    // Command processing
    IF #fbInputs.Cmd_Stop THEN
        // STOP: controlled stop without generating an error + return to safe position
        #bPauseActive := FALSE;
        #bStartSeq := FALSE;
        // Drop every other axis-motion trigger before handing the axes to the STOPPING
        // park move. Without this, a Stop pressed during a clearance/park move (13/16) or
        // during the homing sequence (15) leaves fbMoveX/Z_HomeClr or fbHomeX/Z/Tool
        // executing while fbMoveX/Z_Stop is also commanded -- two MC_ function blocks
        // fighting for the same axis. Latent before the sheet-load park change; state 16
        // is now on the normal cycle path (every reposition), so it is reachable in
        // routine operation rather than only mid-homing.
        #bHomeClrX := FALSE; #bHomeClrZ := FALSE;
        #bHomeXExec := FALSE; #bHomeZExec := FALSE; #bHomeToolExec := FALSE;
        #homeSeqState := 0;
        // If running, go to special STOP sequence; otherwise go directly to STOPPED
        IF (#State >= STATE_STARTING AND #State < STATE_ERROR AND #State <> 100) OR (#State = STATE_PAUSED) THEN
            #State := STATE_STOPPING;
        ELSE
            #State := STATE_STOPPED;
        END_IF;
    END_IF;
    // Reset and Restart are blocked while E-Stop is active.
    // Operator must physically release E-Stop before clearing any error state.
    IF #fbInputs.Cmd_Reset AND (#EStop_OK OR "DB_HMI".Bypass_EStop) THEN
        #bDoHardReset := TRUE;
    END_IF;

    // Btn_Restart - restart program from beginning (from ERROR or PAUSED).
    // This block fires BEFORE the CASE state machine, so CASE 999/25 restart handlers
    // are bypassed. All required cleanup must be done here.
    IF #restartEdge AND (#State = STATE_ERROR OR #State = STATE_PAUSED)
       AND (#EStop_OK OR "DB_HMI".Bypass_EStop) THEN
        #State := STATE_STOPPED;
        #bPauseActive := FALSE;
        #Error := FALSE;
        #bResetRecipe := TRUE;      // Reset recipe handler to IDLE (was missing -- bug fix)
        #prevSafetyError := FALSE;  // Fresh safety evaluation on restart
        #savedLineIndex := -1;
        #savedProgram := -1;
        "DB_HMI".ResumeLine := -1;
        IF NOT "DB_MachineConfig".Bypass_MandrelLock THEN
            #bMandrelRetractPending := TRUE;  // ITEM-32: deferred — spindle may still be spinning; wait SpindleStopSafeTime
        END_IF;
        #fbAlarmManager(NewError := FALSE, NewErrorCode := 0,
                        AcknowledgeError := TRUE);  // Clear active alarm (was missing -- bug fix)
    END_IF;

    // Pause - one-shot SET only (no toggle). Only Btn_Continue resumes.
    IF #fbInputs.Cmd_Pause AND #Running AND NOT #bPauseActive THEN #bPauseActive := TRUE; END_IF;

    #Running := (#State >= 10) AND (#State < STATE_ERROR);
    #IsPaused := (#State = STATE_PAUSED);

    // Update HMI status lamps
    "DB_HMI".IsRunning := #Running;
    "DB_HMI".IsPaused := #IsPaused;
    "DB_HMI".HasError := (#State = STATE_ERROR);

    // Warning: only E-Stop bypass is shown on HMI (Door/Air/Drive bypasses silently permitted for setup)
    // Since 2026-08-12 the bypass no longer blocks auto start, so this banner is the
    // ONLY indication that the machine will run with the E-Stop circuit defeated.
    // WarningID stays 1 (WinCC text list key); the wording changed -- keep
    // tools/hmi_texts.csv row 'warning,1' in step with this string.
    // Priority chain, highest first. E-Stop bypass is never suppressed by anything --
    // it is the only sign that the machine will run unguarded, so it outranks a
    // transient interlock message. A blocked tool jog therefore shows no banner while
    // the bypass is on; the jog is still refused, which is the part that matters.
    "DB_HMI".HasWarning := "DB_HMI".Bypass_EStop OR #bToolAxisBlocked
                           OR #bToolStepBlocked OR #bBlindMoveBlocked;
    IF "DB_HMI".Bypass_EStop THEN
        "DB_HMI".WarningText    := 'DANGER: E-Stop bypassed - machine runs unguarded';
        "DB_HMI".WarningID      := 1;
    ELSIF #bToolAxisBlocked OR #bToolStepBlocked THEN
        // Shown as soon as the tool axis is selected with the lock engaged, not only
        // after a button press: the operator learns why before pushing, and the
        // message explains the refusal if they push anyway. No latch, no timer --
        // it clears itself when the lock releases or another axis is selected.
        // The turret-step buttons (#bToolStepBlocked) have no "selection" to hook, so
        // for them the banner is necessarily press-driven and shares WarningID 3 --
        // same cause, same wording, no new text-list row needed.
        "DB_HMI".WarningText    := 'Tool axis locked - ToolHeadLock is engaged';
        "DB_HMI".WarningID      := 3;
    ELSIF #bBlindMoveBlocked THEN
        // ITEM-56d: MoveAbsolute / GoSafe / GoZero are refused while halted in a PNP zone.
        // A dead button with no explanation is how an operator concludes the panel is broken,
        // so say why and name the two things that DO work. Warning, not an error -- a refused
        // button must never demand a Reset (same rule as the ToolHeadLock interlock above).
        // #bBlindMoveBlocked is assigned near the bottom of this FB, so this reads the previous
        // scan's value; harmless, because STATE_PNP_HALT is held for many scans.
        "DB_HMI".WarningText    := 'Blocked in proximity zone - use jog or Home to escape';
        "DB_HMI".WarningID      := 4;
    ELSE
        "DB_HMI".WarningText    := '';
        "DB_HMI".WarningID      := 0;
    END_IF;

    // Update HMI status message based on state (English only since 2026-08-10 --
    // Spanish comes from a WinCC text list keyed off DB_HMI.MachineState, ITEM-55)
    CASE #State OF
        0:   "DB_HMI".StatusMsg := 'Stopped';
        5:   "DB_HMI".StatusMsg := 'Manual Mode';
        10:  "DB_HMI".StatusMsg := 'Starting...';
        11:  "DB_HMI".StatusMsg := 'Loading recipe...';
        12:  "DB_HMI".StatusMsg := 'Pre-scanning...';
        13:  "DB_HMI".StatusMsg := 'Clearing PNP zone...';
        14:  "DB_HMI".StatusMsg := 'Waiting for sheet...';
        15:  "DB_HMI".StatusMsg := 'Homing...';
        16:  "DB_HMI".StatusMsg := 'Sheet-load park move...';
        17:  "DB_HMI".StatusMsg := 'Lock engaging...';
        18:  "DB_HMI".StatusMsg := 'Stopping...';
        29:  "DB_HMI".StatusMsg := 'Lock releasing...';
        19:  "DB_HMI".StatusMsg := 'Homing (post-stop)...';
        20:  "DB_HMI".StatusMsg := 'Running';
        21:  "DB_HMI".StatusMsg := 'Returning to zero...';
        22:  "DB_HMI".StatusMsg := 'PNP Halt - jog to escape limit zone';
        25:  "DB_HMI".StatusMsg := 'Paused';
        30:  "DB_HMI".StatusMsg := 'Tool Change';
        35:  "DB_HMI".StatusMsg := 'Tool Change Wait';
        100: "DB_HMI".StatusMsg := 'Program Complete';
        999: "DB_HMI".StatusMsg := 'ERROR';
    END_CASE;

    // =========================================================================
    // ALARM MANAGER - call FIRST so outputs are ready for DB_HMI
    // =========================================================================
    // NOTE: Acknowledge is done only on edge (ackEdge), not level.
    // This keeps ActiveError/HMI bools visible until the operator actually presses Ack.
    //
    // Error_ProcessState: captured HERE, guarded, and nowhere else (2026-08-17). It used
    // to be assigned #State unconditionally a few lines below, every scan -- which made it
    // a duplicate of DB_Diagnostic.Process_State and destroyed the thing it was named for.
    // Every diagnostic doc read it as "the state the machine was in when it faulted"; it
    // never held that. One guard here covers all ~30 alarm sites, because they all funnel
    // through #newErrorFlag. Do not add a second writer -- the two that existed
    // (STATE_ERROR in this file, FB_RecipeHandler state 999) both wrote a constant.
    IF #newErrorFlag THEN
        "DB_Diagnostic".Error_ProcessState := #State;
    END_IF;

    #fbAlarmManager(NewError         := #newErrorFlag,
                    NewErrorCode     := #newErrorCode,
                    AcknowledgeError := #ackEdge OR #fbInputs.Cmd_Reset,
                    ActiveProgram    := #activeProgram,
                    ActiveLine       := #fbRecipeHandler.CurrentLine);  // ITEM-26
    #newErrorFlag := FALSE;

    // Debug helpers: copy alarm/diagnostic info into DB_Diagnostic for easy tracing
    // This ensures a snapshot of the latest active error code is always visible for debugging.
    // (Error_ProcessState is NOT written here any more -- see the guarded capture above.
    //  The live state is DB_Diagnostic.Process_State, written at the bottom of this FB.)
    "DB_Diagnostic".Error_Code := #fbAlarmManager.ActiveErrorCode;
    // If recipe reported a line error, keep that; otherwise -1
    IF "DB_Diagnostic".Error_Line < 0 THEN
        "DB_Diagnostic".Error_Line := -1;
    END_IF;

    // Copy alarm outputs to HMI (now reads CURRENT scan values)
    "DB_HMI".ErrorID       := #fbAlarmManager.ActiveErrorCode;
    "DB_HMI".ErrorText     := #fbAlarmManager.ActiveErrorText;
    // ITEM-08: If no active alarm text but a safety condition is blocking, show it.
    // This covers the case where the operator is in STOPPED state with door open / E-Stop active
    // after a previous error was acknowledged — AlarmManager cleared its text but the safety
    // condition is still live and writing to DB_Diagnostic.Error_Text.
    // Use compact customer-facing text here; DB_Diagnostic keeps the developer detail.
    // ITEM-16: ErrorDetail is also written here so the operator does not need DB_Diagnostic.
    IF "DB_HMI".ErrorText = '' AND NOT #fbSafetyMonitor.SafeToRun THEN
        CASE #fbSafetyMonitor.ErrorCode OF
            16#0401: "DB_HMI".ErrorText      := 'EMERGENCY STOP active';
                     "DB_HMI".ErrorDetail    := 'Check E-Stop pushbutton and wiring';
            16#0402: "DB_HMI".ErrorText      := 'Safety door open';
                     "DB_HMI".ErrorDetail    := 'Close the safety door to continue';
            16#0403: "DB_HMI".ErrorText      := 'Drives not ready';
                     "DB_HMI".ErrorDetail    := 'Check contactor, enable wiring and drive status';
            16#0404: "DB_HMI".ErrorText      := 'Air pressure low';
                     "DB_HMI".ErrorDetail    := 'Check air compressor and pressure switch';
            ELSE:    "DB_HMI".ErrorText      := 'Safety interlock active';
                     "DB_HMI".ErrorDetail    := '';
        END_CASE;
    END_IF;
    "DB_HMI".CurrentTool := #CurrentTool;

    // Reset TO errors (only on AckError or full reset)
    // BUG FIX: MC_Reset is triggered only by edge signals. Btn_AckError level signal
    // is not used -- when the button is held, Execute stays HIGH continuously, which
    // adversely affects TO error management (new errors may be masked).
    #fbResetX(Execute := #ackEdge OR #fbInputs.Cmd_Reset, Axis := #Axis_X);
    #fbResetZ(Execute := #ackEdge OR #fbInputs.Cmd_Reset, Axis := #Axis_Z);
    #fbResetTool(Execute := #ackEdge OR #fbInputs.Cmd_Reset, Axis := #Axis_Tool);
    #fbResetSpindle(Execute := #ackEdge OR #fbInputs.Cmd_Reset, Axis := #Axis_Spindle);

    // =========================================================================
    // HARD RESET
    // =========================================================================
    // Single place that defines what a full reset clears.
    // Triggered from exactly two places:
    //   1. bInitDone block (first PLC scan after power-up / warm restart)
    //   2. Cmd_Reset handler (operator presses Reset button)
    // Motion-FB execute flags (bHomeXExec, bStopMoveX, etc.) are cleared by the
    // STATE_STOPPED CASE block which runs on this same scan right after this block.
    IF #bDoHardReset THEN
        // Reference validity -- evaluated FIRST, while #State still holds the state the
        // operator pressed Reset in (the assignment below overwrites it).
        //
        // This used to be an unconditional #bRequireHoming := TRUE at the bottom of the block,
        // which made every Reset cost a full homing cycle on the next auto start. Operators
        // press Reset out of habit, often several times, from an idle machine — where nothing
        // has happened that could invalidate the reference. Now only a reset pressed from a
        // state where an axis could have been moving arms the latch, because #bHaltAllAxes
        // above aborts whatever was in progress.
        //
        // WHITELIST, not blacklist: anything not listed counts as "could have been moving", so
        // a state added later fails safe. The three listed states are motionless by definition:
        //   STOPPED (0)  — idle
        //   MANUAL  (5)  — jogging is tracked by the TO, and STATE_STARTING already handles
        //                  "trusted but parked elsewhere" with a park move. An MC_Home aborted
        //                  mid-seek in manual clears StatusBits.HomingDone by itself, and
        //                  bRefTrusted checks that separately
        //   COMPLETE(100)— program finished, axes parked
        // This NEVER clears the latch — only ever sets it — so a homing requirement raised
        // earlier by an E-Stop, a fault or loss of drive power survives any number of resets.
        IF NOT (#State = STATE_STOPPED OR #State = STATE_MANUAL OR #State = 100) THEN
            #bRequireHoming := TRUE;
        END_IF;
        #bHaltAllAxes    := TRUE;   // ITEM-31: abort any in-progress MC_Home before clearing state
        #State           := STATE_STOPPED;
        #Error           := FALSE;
        #bPauseActive    := FALSE;
        #bResumeSpeedup  := FALSE;   // Cancel any pending pause spin-up wait
        #bResumeLockChk  := FALSE;   // Cancel any pending pause lock verification
        #savedLineIndex  := -1;
        #savedProgram    := -1;
        "DB_HMI".ResumeLine := -1;
        #prevSafetyError := FALSE;
        #bResetRecipe                := TRUE;
        #bRecipeLoadExec             := FALSE;  // drop READ_DBL REQ. fbRecipeLoader.Reset is driven
                                                // by bResetRecipe (set TRUE just above) at its call
                                                // site -- NOT by bDoHardReset, which is cleared at
                                                // the end of this block and would never be seen
                                                // there. That Reset also clears LoadedProgram ->
                                                // forces a fresh copy before the next cycle
        #bSheetWaitPhase2            := FALSE;
        #bSheetWaitPhase3            := FALSE;
        IF NOT "DB_MachineConfig".Bypass_MandrelLock THEN
            #bMandrelRetractPending  := TRUE;   // ITEM-32: deferred — machine may have been RUNNING; wait SpindleStopSafeTime
        END_IF;
        #bSheetHolderRetractHold     := TRUE;   // Release sheet holder regardless of which state was active.
                                                // TRUE (not FALSE) is the safe hard-reset default: this latch
                                                // commands the retract, and the blocked centre will otherwise
                                                // hold the piston wherever the fault left it.
                                                // tonSheetHolderHold needs no explicit reset: its IN is this
                                                // latch, so setting it TRUE here restarts the window cleanly.
        // BackSupport end-of-recipe retract (ITEM-41): deliberately NOT reset here, and the edge
        // memory is deliberately NOT seeded here. Same class of exception as
        // #bMandrelRetractPending above -- an in-flight safety motion outlives the reset.
        //
        // Seeding bBSTerminalPrev := TRUE in this block would suppress the retract exactly when
        // it is most needed: a Reset pressed while RUNNING sets State := STOPPED three lines
        // above, so a seeded edge memory sees terminal->terminal, no rising edge fires, and the
        // BackSupport is left frozen wherever the recipe put it. Power-up needs the seed and
        // gets it in the bInitDone first-scan block instead -- that is the only case where
        // State is already STOPPED before this block runs.
        //
        // Clearing bBSEndRetract here would abandon a retract mid-stroke (Reset pressed inside
        // the 2 s window). Letting it run costs nothing: the block at the bottom of this FB
        // drops every coil when its timer expires, and Cmd_Extend is already FALSE by then.
        //
        // Cmd_Retract still has to be dropped if NO window is running -- otherwise a CMD=41 P2
        // latch survives the reset and holds the cylinder retracting.
        IF NOT #bBSEndRetract THEN
            "DB_Cylinder_BackSupport".Cmd_Retract := FALSE;
        END_IF;
        #bWaitingSpindleStop         := FALSE;  // Cancel any pending spindle-stop wait
        #bSandActive                 := FALSE;  // Cancel the end-of-program sanding dwell.
                                                // tonSandDwell needs no explicit reset: its IN
                                                // is this latch, so clearing it resets the timer.
        #capturedSpindleRPM          := 0.0;
        #spindleStopPT               := T#0MS;
        #prevMDIExec                 := FALSE;  // Clear stale MDI edge (button may be held at reset)
        #bMDI_Cmd40Extend            := FALSE;  // Release MDI CMD=40 BackSupport extend latch
        // CMD=41 edge memory: SEED with the live button state, do not clear. Clearing
        // would let a button still held/latched at reset fire a one-shot immediately.
        #prevBtnCmd41Release         := "DB_Manual".Btn_Cmd41_Release;
        #prevBtnCmd41AtmoOff         := "DB_Manual".Btn_Cmd41_AtmoOff;
        #prevBtnCmd41AtmoOn          := "DB_Manual".Btn_Cmd41_AtmoOn;
        // Reference validity is decided at the TOP of this block (it needs the pre-reset
        // #State). Do not re-add an unconditional #bRequireHoming := TRUE here.
        #bDoHardReset                := FALSE;
    END_IF;

    // =========================================================================
    // SHEET-LOAD PARK TARGET -- soft-limit clamped, single source of truth
    // =========================================================================
    // SheetLoadPos_X/Z are commissioning values typed on the HMI, so clamp them to the
    // configured soft limits before they can reach an MC_MoveAbsolute -- a mistyped value
    // must not be able to drive an axis into a limit.
    //
    // Computed BEFORE the state machine so the "am I already parked?" comparison in
    // STATE_STARTING and the move target it hands to STATE_POST_HOME_CLR / STATE_STOPPING
    // are the same number in the same scan. Comparing against the raw config value while
    // moving to the clamped one would make an out-of-range SheetLoadPos re-issue a
    // pointless park move on every cycle.
    // =========================================================================
    #parkTargetX := MIN(IN1 := MAX(IN1 := "DB_MachineConfig".SheetLoadPos_X,
                                   IN2 := "DB_MachineConfig".SoftLimit_MinX),
                        IN2 := "DB_MachineConfig".SoftLimit_MaxX);
    #parkTargetZ := MIN(IN1 := MAX(IN1 := "DB_MachineConfig".SheetLoadPos_Z,
                                   IN2 := "DB_MachineConfig".SoftLimit_MinZ),
                        IN2 := "DB_MachineConfig".SoftLimit_MaxZ);

    // =========================================================================
    // SANDING DWELL TIME + SPEED -- soft-clamped, single source of truth (2026-08-29)
    // =========================================================================
    // DB_MachineConfig.SandTime_s is WHOLE SECONDS as a plain Int, not the Time type the
    // other timers in that DB use. An S7 Time is milliseconds underneath, and this is the
    // one timer an operator retypes at the machine -- "10" has to mean ten seconds in a
    // plain number field, not ten milliseconds. The conversion lives here.
    //
    // Clamped to 0..SAND_TIME_MAX_S (600 s) BEFORE the multiply, which is also what keeps
    // the arithmetic safe: Int tops out at 32767, so an unclamped SandTime_s * 1000 would
    // overflow. Widen to DInt first anyway -- INT_TO_DINT then multiply, never the reverse.
    #sandTimeSec := MIN(IN1 := MAX(IN1 := "DB_MachineConfig".SandTime_s, IN2 := 0),
                        IN2 := SAND_TIME_MAX_S);
    #sandTimePT  := DINT_TO_TIME(INT_TO_DINT(#sandTimeSec) * 1000);

    // DB_MachineConfig.SandSpeed is typed on the HMI, so clamp it to the machine's real
    // spindle limits before it can reach DB_Spindle.Cmd_SetSpeed -- a mistyped value must
    // not be able to command an out-of-range RPM. Same rule as parkTargetX/Z above.
    //
    // Computed HERE, before the state machine, for the same reason the park targets are:
    // STATE_COMPLETE(100) reads this in the same scan it raises #bSpindleStart, and
    // FB_SpindleControl latches the speed on that start edge. Computed after the CASE it
    // would hold the PREVIOUS scan's value -- 0.0 on the first scan after download, which
    // FB_SpindleControl would clamp up to MinSpeed and then hold for the whole dwell.
    // The restart is currently delayed by SpindleDecelTime, which would mask that; do not
    // rely on it and do not move this below the CASE.
    //
    // A SandSpeed of 0 does NOT arrive here as 0 -- MinSpeed wins the MAX. That is why the
    // arming test in STATE_RUNNING checks SandSpeed > 0.0 rather than checking this value.
    #sandSpeedClamped := MIN(IN1 := MAX(IN1 := "DB_MachineConfig".SandSpeed,
                                        IN2 := "DB_Spindle".MinSpeed),
                             IN2 := "DB_Spindle".MaxSpeed);

    // =========================================================================
    // MAIN STATE MACHINE
    // =========================================================================
    CASE #State OF

        // -----------------------------------------------------------------
        // === STATE_STOPPED (0) ===
        // -----------------------------------------------------------------
        0: // STOPPED
            #StatusID := 0; #bStartSeq := FALSE; #bPreScanExec := FALSE;
            #bRecipeLoadExec := FALSE;   // no recipe copy may stay in flight while idle
            // ITEM-34 FIX: clear only when no safety condition is blocking a start.
            // The ITEM-08 fallback (runs BEFORE this CASE) writes the door-open /
            // E-Stop / air-pressure hint into ErrorText when SafeToRun is FALSE;
            // clearing unconditionally here erased that hint every scan, so the
            // operator saw a machine that refused to start with no explanation.
            IF #fbSafetyMonitor.SafeToRun THEN
                "DB_HMI".ErrorText      := '';
                "DB_HMI".ErrorDetail    := '';
            END_IF;
            // Clear ALL motion-FB execute flags every scan while stopped.
            // Every path that reaches STATE_STOPPED (Cmd_Reset, Ack, Continue,
            // Restart, normal stop sequence) therefore clears these automatically.
            // Without this, a flag stuck TRUE (e.g. bHomeXExec after a homing error)
            // keeps its MC_ FB running → error re-triggers immediately after reset.
            #bHomeXExec    := FALSE; #bHomeZExec    := FALSE; #bHomeToolExec := FALSE;
            #homeSeqState  := 0;
            #bToolExecute  := FALSE;
            #bStopMoveX    := FALSE; #bStopMoveZ    := FALSE;
            #bHomeClrX     := FALSE; #bHomeClrZ     := FALSE;
            #bLockAfterHoming := FALSE;
            // Spindle
            #bSpindleStart       := FALSE;
            #bSpindleStop        := FALSE;
            #bSpindleDecelWait   := FALSE;
            #bSpindlePendingStart := FALSE;
            #bResumeSpeedup      := FALSE;  // Cancel any pending pause spin-up wait
            #bResumeLockChk      := FALSE;  // Cancel any pending pause lock verification
            #bSandActive         := FALSE;  // Cancel the end-of-program sanding dwell. This is
                                            // the Stop-button path: STATE_COMPLETE is excluded
                                            // from the STOPPING branch (see Cmd_Stop handler),
                                            // so Stop during the dwell lands here directly and
                                            // #bSpindleStart above kills the spindle.
            // MandrelLock: clear Cmd_Extend (spring retracts on EStop/power-loss).
            // Cmd_Retract is pulsed by bMandrelRetractPulse (set in STATE_STOPPING only — safe path) to
            // force FB out of State 3 — Mode=0 does not auto-retract on Cmd_Extend=FALSE alone.
            // All other paths (Reset/Error/Complete) use bMandrelRetractPending + tonMandrelRetractWait (ITEM-32).
            "DB_Cylinder_MandrelLock".Cmd_Extend  := FALSE;
            // SheetHolder Cmd_Extend is NOT written here any more: it has a single writer at the
            // bottom of this FB (State = SHEET_WAIT AND NOT Ph3), which drives it FALSE in every
            // other state including this one. Writing it here as well was harmless; writing it
            // NOWHERE on the stop path was the bug -- see the single-writer block for detail.
            // BackSupport: de-energise the atmosphere valve at rest.
            "DB_Cylinder_BackSupport".SolAtmo_Cmd := FALSE;
            // BackSupport extend: clear here too. Previously cleared only by
            // FB_RecipeHandler (RESET / STOP handlers), which left no clear path for
            // the manual CMD=40 button -- it would stay asserted after leaving manual.
            "DB_Cylinder_BackSupport".Cmd_Extend  := FALSE;
            // BackSupport retract: latched by CMD=41 P2 and by the end-of-recipe retract, so it
            // must be dropped while idle -- but ONLY once the end-retract window has finished.
            // Entering STOPPED is exactly what starts that window (bBSEndRetract, block at the
            // bottom of this FB), and this CASE runs every scan, so an unconditional clear here
            // cancelled the retract on the scan it was requested. Gate it on the latch.
            // The end-retract block itself drops Cmd_Retract when its timer expires.
            IF NOT #bBSEndRetract THEN
                "DB_Cylinder_BackSupport".Cmd_Retract := FALSE;
            END_IF;
            // bBSEndRetract / tonBSEndRetract / bBSTerminalPrev are NOT reset here -- see the
            // hard-reset block. Resetting them every idle scan is what kept the end-of-recipe
            // retract from ever firing on a normal stop.
            #bMDI_Cmd40Extend                     := FALSE;  // Drop MDI CMD=40 latch while idle
            // CMD=41 edge memory: track the live button state every scan while idle.
            // STATE_MANUAL is entered only from here (see below), so a button left
            // latched cannot fire a one-shot on the first scan of manual mode.
            #prevBtnCmd41Release := "DB_Manual".Btn_Cmd41_Release;
            #prevBtnCmd41AtmoOff := "DB_Manual".Btn_Cmd41_AtmoOff;
            #prevBtnCmd41AtmoOn  := "DB_Manual".Btn_Cmd41_AtmoOn;

            IF "DB_Manual".ManualModeActive AND #fbSafetyMonitor.SafeToJog THEN
                #State := STATE_MANUAL;
            ELSIF #fbInputs.Cmd_Start AND #SafeToRun THEN
                // Bypass_EStop no longer blocks auto start (2026-08-12). It used to,
                // which made commissioning a running machine without the E-Stop loop
                // impossible. Access control moved to the HMI: the Bypass_EStop switch
                // sits behind a WinCC user authorization, so only a logged-in service
                // user can set it -- the customer's operator account cannot. Do not
                // re-add a NOT Bypass_EStop term here; that would defeat the switch
                // for the service user too. The HasWarning banner stays on the whole
                // time the bypass is set (see the warning block after the CASE).
                //
                // Start pre-scan before running.
                // Always reset fbRecipeHandler here: after any stop or error the handler
                // ends up in STATE_DONE (Done=TRUE). Without this reset, the first scan
                // of RUNNING sees Done=TRUE and immediately reports "recipe complete".
                // (STATE_COMPLETE already does this correctly before its own PRE_SCAN.)
                #bResetRecipe := TRUE;
                #State := STATE_RECIPE_LOAD;   // load recipe out of load memory, then PRE_SCAN
            END_IF;

        // -----------------------------------------------------------------
        // === STATE_MANUAL (5) ===
        // -----------------------------------------------------------------
        5: // MANUAL
            #StatusID := 50;

            // -----------------------------------------------------------------
            // Manual CMD=40 / CMD=41 equivalents (HMI manual page)
            // Each button writes exactly what the matching recipe line writes,
            // so manual and automatic behave identically.
            // Written only here (STATE_MANUAL); STATE_STOPPED and STATE_ERROR
            // drive all three flags FALSE every scan, so nothing can persist
            // after manual mode is left.
            // -----------------------------------------------------------------
            // CMD=40 -- BackSupport extend. Level command: held while the button
            // is held. Releasing mid-stroke returns the FB to idle (blocked
            // centre, cylinder holds position).
            // bMDI_Cmd40Extend is the MDI equivalent: the MDI block below cannot
            // write Cmd_Extend directly, because this line re-evaluates it every
            // scan and would wipe the MDI value one scan later (the cylinder FB
            // then saw a 1-scan pulse and the valve never moved). The MDI sets the
            // latch instead; Param=0 clears it.
            //
            // MDI CMD=40 auto-release -- mirrors FB_RecipeHandler STATE_CYL_GOTO(70) /
            // STATE_CYL_GOTO_WAIT(71): hold Cmd_Extend every scan, then drop it the scan
            // AtSetpoint reports done, or on a cylinder Error. Runs before the assignment
            // below so the release takes effect in the same scan, exactly as state 71 does.
            //
            // Dropping Cmd_Extend does NOT release the cylinder: FB State 3 with
            // PositioningMode=0 holds Sol_A energised (09:833-835) and is left only by
            // Cmd_Retract / Cmd_RetractFull / Cmd_ExtendFull. That is intentional and is
            // the operator's spec -- Sol_A stays ON from CMD=40 through CMD=41 P1, and is
            // released by P2 (Cmd_Retract -> State 2). See the DB_Cylinder_BackSupport
            // header in 02_DataBlocks.scl for the full coil table.
            IF #bMDI_Cmd40Extend THEN
                IF "DB_Cylinder_BackSupport".AtSetpoint THEN
                    #bMDI_Cmd40Extend             := FALSE;
                    // 5, not 1: 'Executed' already uses 1. Two different messages on one
                    // value would collapse into one entry in the HMI text list (ITEM-55).
                    "DB_Manual".MDI_Status        := 5;
                    "DB_Manual".MDI_StatusText    := 'CMD40 done';
                ELSIF "DB_Cylinder_BackSupport".Error THEN
                    #bMDI_Cmd40Extend             := FALSE;
                    "DB_Manual".MDI_Status        := 4;
                    "DB_Manual".MDI_StatusText    := 'CMD40 cylinder error';
                END_IF;
            END_IF;

            "DB_Cylinder_BackSupport".Cmd_Extend := "DB_Manual".Btn_Cmd40_Extend
                                                    OR #bMDI_Cmd40Extend;

            // CMD=41 -- atmosphere overrides. ONE-SHOT (rising edge), exactly like
            // the recipe: FB_RecipeHandler STATE_READ writes these flags on the
            // single scan the line is read and never re-asserts them.
            //
            // Why edge and not level (2026-08-01): these were previously evaluated
            // every scan from latching HMI buttons. A latched button therefore
            // re-wrote its own value continuously and overwrote any later MDI
            // CMD=41 one scan after it was issued -- the operator saw a ~20 ms
            // click on the valve, no state change, and MDI_Status = 'Executed'.
            // With edge detection the button and the MDI write identically: once,
            // per press. AtmoOn -> AtmoOff -> AtmoOn now reproduces P1 -> P2 -> P1,
            // which a latched state cannot express.
            //
            // HMI REQUIREMENT: these three buttons must be MOMENTARY (SetBit on
            // press / ResetBit on release). A latching button fires once per latch
            // cycle and must be un-latched before it can be used again.
            //
            // The safest-first ELSIF order is kept: on a simultaneous press only
            // the safest branch runs, and the other button's edge is consumed by
            // the prev* update below rather than firing on the following scan.
            // Note this no longer forces Sol_B off for as long as Release is held
            // -- with one-shot writes each press acts exactly once.
            IF "DB_Manual".Btn_Cmd41_Release AND NOT #prevBtnCmd41Release THEN      // = CMD=41 Param=3
                "DB_Cylinder_BackSupport".SolAtmo_Cmd := FALSE;
                "DB_Cylinder_BackSupport".Cmd_Retract := FALSE;  // State 2 -> 0: all coils off
            ELSIF "DB_Manual".Btn_Cmd41_AtmoOff AND NOT #prevBtnCmd41AtmoOff THEN   // = CMD=41 Param=2
                "DB_Cylinder_BackSupport".SolAtmo_Cmd := FALSE;
                "DB_Cylinder_BackSupport".Cmd_Retract := TRUE;   // State 3 -> 2: Sol_A off, Sol_B on
            ELSIF "DB_Manual".Btn_Cmd41_AtmoOn AND NOT #prevBtnCmd41AtmoOn THEN     // = CMD=41 Param=1
                "DB_Cylinder_BackSupport".SolAtmo_Cmd := TRUE;   // Sol_A deliberately stays ON
            END_IF;

            // -----------------------------------------------------------------
            // MANUAL MDI -- execute a typed CMD number + Param, once per press.
            //
            // Generic entry point for auxiliary recipe commands. To support a new
            // CMD later, add a branch to the CASE below -- no new DB field and no
            // HMI screen change required.
            //
            // Only auxiliary (non-motion) commands are accepted. Motion commands
            // (CMD=0 / CMD=1) are deliberately rejected: they need feedrate
            // handling and the full soft-limit/motion path. Use Btn_MoveAbsolute
            // for manual positioning instead.
            // -----------------------------------------------------------------
            IF "DB_Manual".Btn_MDI_Execute AND NOT #prevMDIExec THEN
                "DB_Manual".MDI_Status        := 1;              // assume accepted
                "DB_Manual".MDI_StatusText    := 'Executed';
                CASE "DB_Manual".MDI_Cmd OF
                    40: // BackSupport extend -- same sequence as the recipe: assert
                        // Cmd_Extend, hold it, auto-release at AtSetpoint (handled by
                        // the sequencer above).
                        //   Param=1 -> start the extend
                        //   Param=0 -> abort/release early (MDI-only; the recipe ignores
                        //              Param and relies on AtSetpoint alone)
                        IF "DB_Manual".MDI_Param = 1 THEN
                            #bMDI_Cmd40Extend := TRUE;
                        ELSIF "DB_Manual".MDI_Param = 0 THEN
                            #bMDI_Cmd40Extend := FALSE;
                        ELSE
                            "DB_Manual".MDI_Status        := 3;
                            "DB_Manual".MDI_StatusText    := 'CMD40: use Param 0 or 1';
                        END_IF;

                    41: // BackSupport atmosphere / retract -- identical to the recipe CMD=41
                        IF "DB_Manual".MDI_Param = 1 THEN
                            "DB_Cylinder_BackSupport".SolAtmo_Cmd := TRUE;   // Sol_A stays ON
                        ELSIF "DB_Manual".MDI_Param = 2 THEN
                            "DB_Cylinder_BackSupport".SolAtmo_Cmd := FALSE;
                            "DB_Cylinder_BackSupport".Cmd_Retract := TRUE;   // State 3 -> 2
                        ELSIF "DB_Manual".MDI_Param = 3 THEN
                            "DB_Cylinder_BackSupport".SolAtmo_Cmd := FALSE;
                            "DB_Cylinder_BackSupport".Cmd_Retract := FALSE;  // State 2 -> 0
                        ELSE
                            // 6, not 3: CMD40's param error already uses 3 (see above).
                            "DB_Manual".MDI_Status        := 6;
                            "DB_Manual".MDI_StatusText    := 'CMD41: use Param 1,2,3';
                        END_IF;

                    ELSE: // Not an MDI-supported command -- nothing written
                        "DB_Manual".MDI_Status        := 2;
                        "DB_Manual".MDI_StatusText    := 'Unknown/blocked CMD';
                END_CASE;
            END_IF;
            #prevMDIExec := "DB_Manual".Btn_MDI_Execute;
            // CMD=41 button edge memory -- updated after BOTH the button block and
            // the MDI block, so one press is consumed exactly once and the MDI
            // write made this scan survives into the next one.
            #prevBtnCmd41Release := "DB_Manual".Btn_Cmd41_Release;
            #prevBtnCmd41AtmoOff := "DB_Manual".Btn_Cmd41_AtmoOff;
            #prevBtnCmd41AtmoOn  := "DB_Manual".Btn_Cmd41_AtmoOn;

            IF NOT "DB_Manual".ManualModeActive THEN
                // Contactor / enable flags are NOT cleared here any more (2026-08-09).
                //
                // They used to be, "so stale HMI button states cannot activate outputs in
                // STATE_STOPPED" — which only made sense while FC_ContactorControl blocked every
                // output in STOPPED anyway (modePermit, retired with ITEM-49). With that gone,
                // clearing them here physically de-energised the drives on every exit from manual
                // mode, so the axes lost holding torque and their reference every time the
                // operator looked at the manual page. That is one of the "sometimes it homes"
                // paths, and it defeats fast cycle mode after any manual visit.
                //
                // Leaving them as the operator set them is the point: the drives stay powered if
                // they were powered, and if the operator deliberately switched drive power OFF to
                // move an axis by hand, the flags stay FALSE and the reference-validity latch at
                // the bottom of this FB sees it and demands a homing cycle. Either way the
                // behaviour is deterministic. STATE_STARTING forces all of them TRUE on the next
                // auto start regardless.
                //
                // Safety is unchanged: E-Stop (drivePermit in FC_ContactorControl) still drops
                // every contactor and enable output, and nothing here can command motion.
                // Clear MDI result so a stale message does not greet the operator
                // the next time the manual page is opened.
                "DB_Manual".MDI_Status         := 0;
                "DB_Manual".MDI_StatusText     := '';
                #prevMDIExec                   := FALSE;
                #bMDI_Cmd40Extend              := FALSE;  // Do not carry the extend latch out of manual
                // CMD=41 edge memory: seed (not clear) so a button still latched on
                // the way out cannot fire when manual mode is next entered.
                #prevBtnCmd41Release           := "DB_Manual".Btn_Cmd41_Release;
                #prevBtnCmd41AtmoOff           := "DB_Manual".Btn_Cmd41_AtmoOff;
                #prevBtnCmd41AtmoOn            := "DB_Manual".Btn_Cmd41_AtmoOn;
                #State := 0;
            ELSIF #fbInputs.Cmd_Start AND #SafeToRun THEN
                // Bypass_EStop no longer blocks the manual -> auto transition either
                // (2026-08-12) -- same reasoning as the STATE_STOPPED Start handler.
                "DB_Manual".ManualModeActive := FALSE;
                #bResetRecipe := TRUE;  // Same as STATE_STOPPED Cmd_Start handler (see comment there)
                #State := STATE_RECIPE_LOAD;   // load recipe out of load memory, then PRE_SCAN
            END_IF;

        // -----------------------------------------------------------------
        // === STATE_RECIPE_LOAD (11) ===
        // -----------------------------------------------------------------
        // Copy the selected recipe out of LOAD memory into DB_SelectedRecipe
        // before anything reads it. Entered from every path that used to go
        // straight to PRE_SCAN: STOPPED Start, MANUAL Start, COMPLETE
        // restart/Start, COMPLETE Reset.
        //
        // Why this must run EVERY cycle start and not be skipped when the same
        // program is selected again: a recipe re-downloaded from CAM changes the
        // load-memory contents while DB_SelectedRecipe still holds the old data.
        // Skipping the copy would machine the previous geometry with no warning.
        // The copy costs a fraction of a second, once, with the machine standing
        // still -- do not "optimise" it away.
        //
        // The machine is stationary here (same as PRE_SCAN: contactors open,
        // drives not yet enabled), so a few extra scans cost nothing.
        // -----------------------------------------------------------------
        11: // RECIPE LOAD - copy selected recipe from load memory
            #StatusID := 11;
            #bRecipeLoadExec := TRUE;   // level; FB takes the rising edge

            IF #fbRecipeLoader.Error THEN
                // READ_DBL refused the transfer, or it never completed.
                #bRecipeLoadExec := FALSE;
                #newErrorFlag := TRUE;
                // Same pattern as the 16#0310 / 16#0311 sites next door: context goes
                // to DB_Diagnostic.Error_Text, never to DB_HMI.ErrorText (single-writer
                // rule). 16#FFFF here means the watchdog fired, not a READ_DBL code.
                // ErrorPhase (1 = Header, 2 = chunk, 3 = chunk verify, 4 = checksum)
                // says WHICH stage failed -- the 2026-08-06 field fault was a silent
                // Lines failure, so this must stay visible.
                IF #fbRecipeLoader.ErrorPhase = 4 THEN
                    // Phase 4: the copy is COMPLETE and wrong. Every line arrived,
                    // the END marker is where the Header says, and the checksum
                    // still disagrees -- so this is not a transfer fault and must
                    // not be reported as one. Either the recipe DB in load memory
                    // is not the export the CAM computed the checksum over (the
                    // usual cause: 02b imported without re-importing the recipes),
                    // or the two checksum implementations disagree. Both numbers
                    // go in the text, because the pair is what tells them apart.
                    #newErrorCode := 16#0316;
                    "DB_Diagnostic".Error_Text := CONCAT(
                        IN1 := CONCAT(IN1 := 'Recipe checksum mismatch: PLC ',
                                      IN2 := UDINT_TO_STRING(#fbRecipeLoader.ChecksumCalc)),
                        IN2 := CONCAT(IN1 := ' vs CAM ',
                                      IN2 := UDINT_TO_STRING("DB_SelectedRecipe".Header.Checksum)));

                ELSIF #fbRecipeLoader.ErrorPhase = 3 THEN
                    // Phase 3 is NOT a READ_DBL error: every call returned RET_VAL = 0
                    // and the chunk still came back with holes, on every retry. Separate
                    // code so the operator is not sent looking for a transfer fault.
                    // ErrorChunk is the diagnostic that matters: WHICH chunk refuses to
                    // arrive tells us whether the fault is positional (always the same
                    // chunk -> suspect that region of the source DB) or random (-> the
                    // transfer mechanism itself). 0 = the assembled buffer failed its
                    // END-marker cross-check rather than any single chunk.
                    #newErrorCode := 16#0314;
                    "DB_Diagnostic".Error_Text := CONCAT(
                        IN1 := 'Recipe chunk never arrived intact (RET_VAL=0), chunk ',
                        IN2 := INT_TO_STRING(#fbRecipeLoader.ErrorChunk));
                ELSE
                    #newErrorCode := 16#0312;   // Recipe load from load memory failed
                    "DB_Diagnostic".Error_Text := CONCAT(
                        IN1 := CONCAT(IN1 := 'Recipe load failed, phase ',
                                      IN2 := INT_TO_STRING(#fbRecipeLoader.ErrorPhase)),
                        IN2 := CONCAT(IN1 := CONCAT(IN1 := ' (1=Header 2=chunk ',
                                                    IN2 := INT_TO_STRING(#fbRecipeLoader.ErrorChunk)),
                                      IN2 := CONCAT(IN1 := '), RET_VAL=',
                                                    IN2 := INT_TO_STRING(WORD_TO_INT(#fbRecipeLoader.ErrorCode)))));
                END_IF;
                #State := STATE_ERROR;

            ELSIF #fbRecipeLoader.Done THEN
                #bRecipeLoadExec := FALSE;
                "DB_Diagnostic".Recipe_LoadedProgram := #fbRecipeLoader.LoadedProgram;
                #State := STATE_PRE_SCAN;
            END_IF;

        // -----------------------------------------------------------------
        // === STATE_PRE_SCAN (12) ===
        // -----------------------------------------------------------------
        12: // PRE-SCAN - Validate recipe before running
            #StatusID := 12;
            #bPreScanExec := TRUE;
            // Redundant since 2026-07-31 (the flag is now self-cleared after the
            // fbRecipeHandler call each scan); kept as a belt-and-braces clear.
            #bResetRecipe := FALSE;

            // Line count + tool table read from the recipe buffer's Header
            // (both written by the CAM post-processor -- see CAM_TOOL_TABLE_HANDOVER.md).
            // 2026-08-04: was a five-way CASE over DB_RecipeProgram1..5. Those now
            // live in load memory and cannot be read directly; STATE_RECIPE_LOAD(11)
            // has already copied the selected one into DB_SelectedRecipe.
            #activeLineCount    := "DB_SelectedRecipe".Header.LineCount;
            #hdrProvidesToolCfg := "DB_SelectedRecipe".Header.ProvidesToolConfig;
            #hdrToolCount       := "DB_SelectedRecipe".Header.ToolCount;
            #hdrAutoCalc        := "DB_SelectedRecipe".Header.AutoCalcAngles;
            #hdrToolCodes       := "DB_SelectedRecipe".Header.ToolCode_List;
            #hdrToolAngles      := "DB_SelectedRecipe".Header.ToolAngle_List;

            // Validate: 0 = recipe not loaded (Header not written yet).
            // Upper bound is now the ACTUAL array size -- this used to accept up to
            // 999 against an Array[0..349], so a header claiming 400+ lines read past
            // the end of the array. Closed by construction: the guard and the array
            // are both 1000 now. Keep them in step if the array size ever changes.
            // exp/velocity-path-350: guard lowered 1000 -> 400 (2026-09-14), raised to
            // 500 (2026-09-16), together with DB_SelectedRecipe.Lines and LINES_MAX in
            // the loader. The comment above predates this branch.
            // <<< GENERATED:LINECOUNT_GUARD -- do not hand-edit; run tools/gen_recipe_slots.py --lines N >>>
            IF #activeLineCount <= 0 OR #activeLineCount > 800 THEN
            // <<< END GENERATED:LINECOUNT_GUARD >>>
                #newErrorFlag := TRUE;     // BUG FIX: was missing -- alarm manager never latched 16#0310,
                                           // so HMI showed ERROR state with empty text and no history entry
                #newErrorCode := 16#0310;  // Recipe: invalid line count (not loaded?)
                #bPreScanExec := FALSE;    // Do not start a scan on garbage LineCount
                "DB_Diagnostic".Error_Text := 'Recipe not loaded: Header.LineCount invalid';
                // Single-writer: HMI text comes from FB_AlarmManager (CASE 16#0310)
                #State := STATE_ERROR;

            // END-MARKER GUARD (2026-08-06, added after the field fault where the
            // Lines array arrived all zero while the Header was plausible). The
            // recipe format REQUIRES the last line to be CMD=99 (PROGRAM_END --
            // PLC_Recipe_Format_Spec.md, CMD table + template line N-1), and the
            // CAM post-processor always emits it. A buffer whose header claims N
            // lines but whose line N-1 is not 99 is empty or corrupt -- catching
            // it here stops the machine from "running" a program of zero-moves.
            ELSIF "DB_SelectedRecipe".Lines[#activeLineCount - 1].CMD <> 99 THEN
                #newErrorFlag := TRUE;
                #newErrorCode := 16#0313;  // Recipe buffer corrupt: no END marker
                #bPreScanExec := FALSE;
                "DB_Diagnostic".Error_Text := CONCAT(
                    IN1 := 'Recipe buffer corrupt: Lines empty or truncated, last CMD=',
                    IN2 := INT_TO_STRING(BYTE_TO_INT(
                        "DB_SelectedRecipe".Lines[#activeLineCount - 1].CMD)));
                // Single-writer: HMI text comes from FB_AlarmManager (CASE 16#0313)
                #State := STATE_ERROR;
            END_IF;

            // Apply the CAM-authored tool table BEFORE the pre-scan validates tool codes.
            // "Recipe always wins": every recipe must carry its own tool table, else it is
            // rejected here (16#0311). Skipped if the LineCount check already bailed
            // (#bPreScanExec cleared) so we do not overwrite the 16#0310 error.
            IF #bPreScanExec THEN
                IF NOT #hdrProvidesToolCfg THEN
                    #newErrorFlag := TRUE;
                    #newErrorCode := 16#0311;  // Recipe has no tool table (ProvidesToolConfig=FALSE)
                    #bPreScanExec := FALSE;
                    "DB_Diagnostic".Error_Text := 'Recipe missing tool table (ProvidesToolConfig=FALSE)';
                    // Single-writer: HMI text comes from FB_AlarmManager (CASE 16#0311)
                    #State := STATE_ERROR;
                ELSE
                    // Defensive clamp: ToolCode_List / ToolAngle_List are Array[1..4].
                    // A ToolCount > 4 would index out of bounds in the recipe lookup
                    // loops (05_RecipeHandler) -> CPU STOP. Clamp to 1..4 here.
                    IF #hdrToolCount < 1 THEN #hdrToolCount := 1; END_IF;
                    IF #hdrToolCount > 4 THEN #hdrToolCount := 4; END_IF;
                    "DB_MachineConfig".ToolCount   := #hdrToolCount;
                    "DB_ToolConfig".AutoCalcAngles := #hdrAutoCalc;
                    FOR #applyIndex := 1 TO 4 DO
                        "DB_ToolConfig".ToolCode_List[#applyIndex] := #hdrToolCodes[#applyIndex];
                        "DB_HMI".ToolSlotCode[#applyIndex]         := #hdrToolCodes[#applyIndex];  // HMI display mirror
                    END_FOR;
                    // When AutoCalcAngles=FALSE the recipe supplies explicit slot angles.
                    // When TRUE, FC_ToolAngleCalc recomputes them every scan from ToolCount.
                    IF NOT #hdrAutoCalc THEN
                        "DB_ToolConfig".Tool1_Position := #hdrToolAngles[1];
                        "DB_ToolConfig".Tool2_Position := #hdrToolAngles[2];
                        "DB_ToolConfig".Tool3_Position := #hdrToolAngles[3];
                        "DB_ToolConfig".Tool4_Position := #hdrToolAngles[4];
                    END_IF;
                END_IF;
            END_IF;

            // NOTE: fbPreScan is called unconditionally at the bottom of this FB
            // (next to fbRecipeHandler), NOT here. BUG FIX: when it was called only
            // inside this CASE branch, Execute never went FALSE between runs, so the
            // FB stayed latched in its DONE state and every start after the first
            // returned the PREVIOUS run's Valid/bounding-box instantly -- recipe
            // validation was silently skipped from the second cycle onward.

            // Update progress every scan during pre-scan (HMI bar)
            "DB_HMI".PreScanProgress := #fbPreScan.Progress;

            IF #fbPreScan.Done THEN
                #bPreScanExec := FALSE;

                // Update HMI with bounding box
                "DB_HMI".BoundingBox_MinX := #fbPreScan.MinX;
                "DB_HMI".BoundingBox_MaxX := #fbPreScan.MaxX;
                "DB_HMI".BoundingBox_MinZ := #fbPreScan.MinZ;
                "DB_HMI".BoundingBox_MaxZ := #fbPreScan.MaxZ;
                "DB_HMI".BoundingBox_Valid := #fbPreScan.Valid;

                // Update diagnostic
                "DB_Diagnostic".PreScan_Complete := TRUE;
                "DB_Diagnostic".PreScan_Valid := #fbPreScan.Valid;
                "DB_Diagnostic".PreScan_ErrorLine := #fbPreScan.ErrorLine;

                IF #fbPreScan.Valid THEN
                    #State := STATE_STARTING;
                ELSE
                    // Pre-scan failed - limits exceeded.
                    // Single-writer: report via queue so the failing line number reaches the
                    // displayed text (queue path shows Details as the EN ErrorText; ES comes
                    // from the FB_AlarmManager CASE table for 16#0305).
                    "FC_ReportError"(Code := 16#0305,
                                     Details := CONCAT(IN1 := 'PreScan Ln', IN2 := CONCAT(
                                                IN1 := INT_TO_STRING(#fbPreScan.ErrorLine), IN2 := CONCAT(
                                                IN1 := ': ', IN2 := #fbPreScan.ErrorDesc))),
                                     Source := 'Recipe');
                    "DB_HMI".ErrorDetail    := CONCAT(IN1 := 'Check line ', IN2 := INT_TO_STRING(#fbPreScan.ErrorLine));
                    "DB_Diagnostic".Error_Text := CONCAT(IN1 := 'PreScan failed Ln',
                                                  IN2 := CONCAT(IN1 := INT_TO_STRING(#fbPreScan.ErrorLine),
                                                  IN2 := CONCAT(IN1 := ': ', IN2 := #fbPreScan.ErrorDesc)));
                    #State := STATE_ERROR;
                END_IF;
            END_IF;

        // -----------------------------------------------------------------
        // === STATE_STARTING (10) ===
        // -----------------------------------------------------------------
        10: // STARTING
            #StatusID := 1;
            // Auto-enable drives for auto mode -- contactors and enable signals are set automatically.
            // In manual mode (STATE_MANUAL) they are under HMI control; PLC takes over when switching to auto.
            "DB_HMI".Btn_Contactor_X       := TRUE;
            "DB_HMI".Btn_Contactor_Z       := TRUE;
            "DB_HMI".Btn_Contactor_Tool    := NOT "DB_MachineConfig".Bypass_ToolAxis;
            "DB_HMI".Btn_Contactor_Spindle := NOT "DB_HMI".Bypass_Spindle;
            "DB_HMI".Btn_Enable_X          := TRUE;
            "DB_HMI".Btn_Enable_Z          := TRUE;
            // Tool enable (2026-08-16, %Q8.1). Same drive model as X/Z, so treated identically:
            // asserted in the same scan as its contactor, no settle delay. What fixes the 16#000D
            // suspect is that this output is LOW from power-up until Start -- previously the tool
            // had no enable output and the drive's enable was held on locally, so the servo came
            // up already enabled the instant its contactor closed.
            // No Bypass_ToolAxis term needed: FC_ContactorControl ANDs the output with
            // Btn_Contactor_Tool, which is already FALSE when the axis is bypassed.
            "DB_HMI".Btn_Enable_Tool       := TRUE;
            //
            // Wait for all drives to report ready before issuing any motion command.
            // Physical contactor close + drive boot can take up to several hundred ms.
            // tonDriveReady is called unconditionally near the timer section (auto-resets on exit).
            //
            // The tool term was added 2026-08-16 with the %Q8.1 enable output. Before that the
            // machine confirmed X and Z were up and then started moving without ever checking
            // the tool drive -- so a tool drive that failed to come up was found later, as a
            // homing or motion failure, instead of here as 16#000C. Bypass_ToolAxis drops the
            // term because with the bypass set Btn_Contactor_Tool is FALSE by design, so
            // fbPowerTool.Status can never come TRUE and the start would hang to timeout.
            IF #fbPowerX.Status AND #fbPowerZ.Status
               AND (#fbPowerTool.Status OR "DB_MachineConfig".Bypass_ToolAxis) THEN
                // Drives ready -- three-way decision: home, reposition, or load the sheet.
                //
                // The axis reference is TRUSTED only when every required axis reports
                // HomingDone AND nothing has invalidated it since the last completed
                // homing cycle (bRequireHoming: E-Stop, STATE_ERROR, hard reset, power-up).
                // StatusBits.HomingDone alone is not enough -- whether the TO clears it
                // when MC_Power drops is encoder-type dependent, and an open-loop axis can
                // lose steps during an E-Stop while still reporting HomingDone=TRUE.
                #bRefTrusted := #Axis_X.StatusBits.HomingDone
                                AND #Axis_Z.StatusBits.HomingDone
                                AND (#Axis_Tool.StatusBits.HomingDone
                                     OR "DB_MachineConfig".Bypass_ToolAxis)
                                AND NOT #bRequireHoming;

                IF NOT #bRefTrusted OR "DB_MachineConfig".AlwaysHomeOnAutoStart THEN
                    // (1) Reference suspect, or the operator forced homing on every cycle.
                    // Full reference seek. NEVER command an absolute move here -- the
                    // coordinate system cannot be trusted until MC_Home completes.
                    // If in PNP zone, clear it first (target = legacy PNP escape position).
                    #bHomeClrX := #HW_PNP_X_Min AND NOT #Axis_X.StatusBits.HomingDone;
                    #bHomeClrZ := #HW_PNP_Z_Min AND NOT #Axis_Z.StatusBits.HomingDone;
                    IF #bHomeClrX OR #bHomeClrZ THEN
                        #clrTargetX  := "DB_MachineConfig".HomeOffset_X + "DB_MachineConfig".PostHome_Clearance;
                        #clrTargetZ  := "DB_MachineConfig".HomeOffset_Z + "DB_MachineConfig".PostHome_Clearance;
                        #clrVelocity := "DB_MachineConfig".HomeVelocity;  // slow: escaping a PNP sensor un-homed
                        #State := STATE_PRE_HOME_CLR;
                    ELSE
                        #homeSeqState := 1;
                        #bHomeXExec := TRUE; #bHomeZExec := FALSE;
                        #State := STATE_HOMING;
                    END_IF;
                ELSIF ABS(#Axis_X.ActualPosition - #parkTargetX) > "DB_MachineConfig".SheetLoadTol
                   OR ABS(#Axis_Z.ActualPosition - #parkTargetZ) > "DB_MachineConfig".SheetLoadTol THEN
                    // (2) Reference trusted but the axes are parked somewhere else -- e.g.
                    // the operator jogged in MANUAL between parts, or the last run was
                    // aborted. Reposition to the sheet-load park instead of paying for a
                    // full homing cycle. Safe: the reference is valid, the move is a normal
                    // absolute move, and the target is clamped to the soft limits.
                    // STATE_POST_HOME_CLR already does "move X+Z to target, then SHEET_WAIT".
                    #bHomeClrX   := TRUE; #bHomeClrZ := TRUE;
                    #clrTargetX  := #parkTargetX;
                    #clrTargetZ  := #parkTargetZ;
                    #clrVelocity := "DB_MachineConfig".RapidVelocity;  // can be a long travel -- not the 5 mm/s clearance speed
                    #State       := STATE_POST_HOME_CLR;
                ELSE
                    // (3) Reference trusted AND already parked at the sheet-load position:
                    // no motion needed -- straight to sheet insertion. This is the fast
                    // path that removes the homing seek from every cycle after the first.
                    // NOTE: goes to SHEET_WAIT, never straight to LOCK_EXTEND_WAIT -- the
                    // operator must still load a sheet and the MandrelLock must still clamp
                    // (both were released at the end of the previous cycle).
                    #bSheetWaitPhase2 := FALSE;
                    #bSheetWaitPhase3 := FALSE;
                    #State := STATE_SHEET_WAIT;
                END_IF;
            ELSIF #tonDriveReady.Q THEN
                // Timeout: drives did not become ready within Timeout_DriveReady.
                // Name the offender -- with three axes in the test, 'a drive' is not actionable.
                #newErrorFlag := TRUE;
                #newErrorCode := 16#000C;
                IF NOT #fbPowerX.Status THEN
                    "DB_HMI".ErrorDetail := 'X drive not ready - contactor closed but no enable/ready';
                ELSIF NOT #fbPowerZ.Status THEN
                    "DB_HMI".ErrorDetail := 'Z drive not ready - contactor closed but no enable/ready';
                ELSE
                    "DB_HMI".ErrorDetail := 'Tool drive not ready - check %Q8.1 enable and contactor';
                END_IF;
                "DB_Diagnostic".Error_Text := "DB_HMI".ErrorDetail;
                #State := STATE_ERROR;
            END_IF;

        // -----------------------------------------------------------------
        // === STATE_HOMING (15) ===
        // -----------------------------------------------------------------
        15: // HOMING (sequential: X then Z in active homing mode 3)
            #StatusID := 2;
            // Ensure other stop/homing triggers are not interfering
            IF #homeSeqState = 1 THEN
                // Homing X
                #bHomeXExec := TRUE;
                #bHomeZExec := FALSE;
                IF #fbHomeX.Done THEN
                    #bHomeXExec := FALSE;
                    #homeSeqState := 2;    // proceed to homing Z
                    #bHomeZExec := TRUE;
                ELSIF #fbHomeX.Error THEN
                    #bHomeXExec := FALSE;
                    #bHomeZExec := FALSE;
                    #State := STATE_ERROR;
                    #newErrorFlag := TRUE;
                    #newErrorCode := 16#0003;
                    "DB_Diagnostic".HomeX_ErrorID := #fbHomeX.ErrorID;
                    "DB_Diagnostic".TO_ErrorText  := "FC_TO_ErrorText"(Code := #fbHomeX.ErrorID);
                    "DB_HMI".ErrorDetail    := CONCAT(IN1 := 'TO:', IN2 := "DB_Diagnostic".TO_ErrorText);
                END_IF;
            ELSIF #homeSeqState = 2 THEN
                // Homing Z
                #bHomeXExec := FALSE;
                #bHomeZExec := TRUE;
                IF #fbHomeZ.Done THEN
                    #bHomeZExec := FALSE;
                    IF NOT "DB_MachineConfig".Bypass_ToolAxis THEN
                        // Proceed to tool axis homing (step 3)
                        #homeSeqState := 3;
                        #bHomeToolExec := TRUE;
                    ELSE
                        // Tool axis bypassed -- go to post-homing park move.
                        // Target is the sheet-load park, not HomeOffset + PostHome_Clearance:
                        // the machine parks at ONE position for sheet loading on every path.
                        #homeSeqState := 0;
                        #bHomeClrX := TRUE; #bHomeClrZ := TRUE;
                        #clrTargetX  := #parkTargetX;
                        #clrTargetZ  := #parkTargetZ;
                        #clrVelocity := "DB_MachineConfig".RapidVelocity;
                        #CurrentTool := 1;  // Tool axis homed to slot 1 position
                        #bRequireHoming := FALSE;  // Reference re-established -- trust it again
                        #State := STATE_POST_HOME_CLR;
                    END_IF;
                ELSIF #fbHomeZ.Error THEN
                    #bHomeZExec := FALSE;
                    #State := STATE_ERROR;
                    #newErrorFlag := TRUE;
                    #newErrorCode := 16#0004;
                    "DB_Diagnostic".HomeZ_ErrorID := #fbHomeZ.ErrorID;
                    "DB_Diagnostic".TO_ErrorText  := "FC_TO_ErrorText"(Code := #fbHomeZ.ErrorID);
                    "DB_HMI".ErrorDetail    := CONCAT(IN1 := 'TO:', IN2 := "DB_Diagnostic".TO_ErrorText);
                END_IF;
            ELSIF #homeSeqState = 3 THEN
                // Homing Tool axis
                #bHomeToolExec := TRUE;
                IF #fbHomeTool.Done THEN
                    #bHomeToolExec := FALSE;
                    #homeSeqState := 0;
                    // Tool done -- proceed to the post-homing park move for X and Z.
                    // Target is the sheet-load park, not HomeOffset + PostHome_Clearance:
                    // the machine parks at ONE position for sheet loading on every path.
                    #bHomeClrX := TRUE; #bHomeClrZ := TRUE;
                    #clrTargetX  := #parkTargetX;
                    #clrTargetZ  := #parkTargetZ;
                    #clrVelocity := "DB_MachineConfig".RapidVelocity;
                    #CurrentTool := 1;  // Tool axis homed to slot 1 position
                    #bRequireHoming := FALSE;  // Reference re-established -- trust it again
                    #State := STATE_POST_HOME_CLR;
                ELSIF #fbHomeTool.Error THEN
                    #bHomeToolExec := FALSE;
                    #State := STATE_ERROR;
                    #newErrorFlag := TRUE;
                    #newErrorCode := 16#0007;
                    "DB_Diagnostic".HomeTool_ErrorID := #fbHomeTool.ErrorID;
                    "DB_Diagnostic".TO_ErrorText     := "FC_TO_ErrorText"(Code := #fbHomeTool.ErrorID);
                    "DB_HMI".ErrorDetail    := CONCAT(IN1 := 'TO:', IN2 := "DB_Diagnostic".TO_ErrorText);
                END_IF;
            ELSE
                // Fallback: if homeSeqState not set, go to STARTING check
                #homeSeqState := 0;
                #State := STATE_STARTING;
            END_IF;
            // Homing timeout: X+Z+Tool combined must complete within 120s
            IF #tonHomingTimeout.Q THEN
                #bHomeXExec := FALSE;
                #bHomeZExec := FALSE;
                #bHomeToolExec := FALSE;
                #homeSeqState := 0;
                #State := STATE_ERROR;
                #newErrorFlag := TRUE;
                #newErrorCode := 16#000B;
                "DB_HMI".ErrorDetail    := 'Homing did not complete - check reference switch/drive';
            END_IF;

        // -----------------------------------------------------------------
        // === STATE_PRE_HOME_CLR (13) ===
        // -----------------------------------------------------------------
        13: // PRE_HOME_CLR -- Clear PNP zone before homing
            #StatusID := 2;
            // Transition to homing as soon as clearance move finishes
            IF (NOT #bHomeClrX OR #fbMoveX_HomeClr.Done) AND (NOT #bHomeClrZ OR #fbMoveZ_HomeClr.Done) THEN
                #bHomeClrX := FALSE; #bHomeClrZ := FALSE;
                #homeSeqState := 1; #bHomeXExec := TRUE; #bHomeZExec := FALSE;
                #State := STATE_HOMING;
            ELSIF (#bHomeClrX AND #fbMoveX_HomeClr.Error) OR (#bHomeClrZ AND #fbMoveZ_HomeClr.Error) THEN
                #bHomeClrX := FALSE; #bHomeClrZ := FALSE;
                // Single-writer: queue path keeps the clearance-move context in the displayed text
                "FC_ReportError"(Code := 16#0001,
                                 Details := 'Pre-home clearance move failed - axis could not clear PNP zone',
                                 Source := 'Process');
                "DB_HMI".ErrorDetail    := 'Axis could not clear PNP zone before homing - check drive';
                #State := STATE_ERROR;
            END_IF;

        // -----------------------------------------------------------------
        // === STATE_POST_HOME_CLR (16) ===
        // Move X and Z to #clrTargetX/Z, then hand over to SHEET_WAIT.
        // Two entry paths, same behaviour -- both target the sheet-load park:
        //   • from STATE_HOMING       -- after a completed reference seek
        //   • from STATE_STARTING (2) -- reference trusted but axes parked elsewhere
        // -----------------------------------------------------------------
        16: // POST_HOME_CLR -- Move X and Z to the sheet-load park position
            #StatusID := 2;
            IF (NOT #bHomeClrX OR #fbMoveX_HomeClr.Done) AND (NOT #bHomeClrZ OR #fbMoveZ_HomeClr.Done) THEN
                #bHomeClrX := FALSE; #bHomeClrZ := FALSE;
                // Parked: wait for sheet insertion before engaging ToolHeadLock
                #bSheetWaitPhase2 := FALSE;  // Always start in phase 1 (show prompt)
                #bSheetWaitPhase3 := FALSE;  // Phase 3 must not survive from an aborted cycle
                #State := STATE_SHEET_WAIT;
            ELSIF (#bHomeClrX AND #fbMoveX_HomeClr.Error) OR (#bHomeClrZ AND #fbMoveZ_HomeClr.Error) THEN
                #bHomeClrX := FALSE; #bHomeClrZ := FALSE;
                // Single-writer: queue path keeps the clearance-move context in the displayed text
                "FC_ReportError"(Code := 16#0001,
                                 Details := 'Park move failed - axis could not reach sheet-load position',
                                 Source := 'Process');
                "DB_HMI".ErrorDetail    := 'Axis could not reach sheet-load position - check drive/SheetLoadPos';
                #State := STATE_ERROR;
            END_IF;

        // -----------------------------------------------------------------
        // === STATE_SHEET_WAIT (14) ===
        // Phase 1: SheetHolder extends to hold the form; HMI prompt; wait operator
        //          both-button confirm (Cmd_Start rising edge).
        // Phase 2: MandrelLock extends (open-loop T#5S) to clamp the mandrel.
        // Phase 3: SheetHolder retracts (open-loop T#5S) to clear; then → LOCK_EXTEND_WAIT
        //          so ToolHeadLock engages before RUNNING.
        // -----------------------------------------------------------------
        14: // SHEET_WAIT
            #StatusID := 14;
            IF NOT #bSheetWaitPhase2 AND NOT #bSheetWaitPhase3 THEN
                // Phase 1: extend SheetHolder and prompt operator to insert the sheet.
                // Drop any retract hold left over from the previous cycle first -- the FB
                // gives Cmd_Extend priority anyway, but leaving both asserted is confusing
                // to read online and pointless once we are commanding the other direction.
                // Cmd_Extend itself is driven by the single writer at the bottom of this FB
                // (TRUE while State = SHEET_WAIT AND NOT Ph3).
                #bSheetHolderRetractHold := FALSE;
                "DB_HMI".HasWarning     := TRUE;
                "DB_HMI".WarningText    := 'Insert sheet, then press both start buttons';
                "DB_HMI".WarningID      := 2;
                IF #fbInputs.Cmd_Start THEN
                    // Operator confirmed — clear prompt
                    "DB_HMI".HasWarning     := FALSE;
                    "DB_HMI".WarningText    := '';
                    "DB_HMI".WarningID      := 0;
                    IF NOT "DB_MachineConfig".Bypass_MandrelLock THEN
                        // Normal: extend MandrelLock (Ph2), then SheetHolder retracts (Ph3)
                        "DB_Cylinder_MandrelLock".Cmd_Extend := TRUE;
                        #bSheetWaitPhase2 := TRUE;
                    ELSE
                        // Bypass: no MandrelLock cylinder — skip Ph2, go straight to Ph3 (SheetHolder retract).
                        // Setting Ph3 also drops Cmd_Extend via the single writer at the bottom of this FB.
                        #bSheetHolderRetractHold := TRUE;
                        #bSheetWaitPhase3 := TRUE;
                    END_IF;
                END_IF;
            ELSIF #bSheetWaitPhase2 THEN
                // Phase 2: open-loop wait T#5S for MandrelLock full stroke
                // tonMandrelWait is driven by the global timer section below (IN when state=14 AND phase2)
                IF #tonMandrelWait.Q THEN
                    // MandrelLock assumed clamped — retract SheetHolder.
                    // Ph3 drops Cmd_Extend via the single writer at the bottom of this FB.
                    #bSheetHolderRetractHold := TRUE;   // Hold Cmd_Retract → Sol_B drives the piston back
                    #bSheetWaitPhase2 := FALSE;
                    #bSheetWaitPhase3 := TRUE;
                END_IF;
            ELSE
                // Phase 3: open-loop wait T#5S for SheetHolder to fully retract
                // tonSheetHolderRetract driven by global timer section below (IN when state=14 AND phase3)
                IF #tonSheetHolderRetract.Q THEN
                    #State := STATE_LOCK_EXTEND_WAIT;  // ToolHeadLock engages, then → RUNNING
                END_IF;
            END_IF;

        // -----------------------------------------------------------------
        // === STATE_RUNNING (20) ===
        // -----------------------------------------------------------------
        20: // RUNNING
            #StatusID := 3; #bStartSeq := TRUE;
            #timerRunning := TRUE;  // Start cycle timer

            // Update HMI
            "DB_HMI".CurrentLine := #fbRecipeHandler.CurrentLine;
            "DB_HMI".ProgressPercent := #fbRecipeHandler.Progress;
            "DB_HMI".FeedrateActive := #fbRecipeHandler.ActiveFeedrate;

            IF #bPauseActive THEN #State := STATE_PAUSED; END_IF;

            // Tool change request (bypass if no tool axis)
            IF #fbRecipeHandler.ToolChangeReq THEN
                IF "DB_MachineConfig".Bypass_ToolAxis THEN
                    // Skip tool change - clear request and continue
                    #fbRecipeHandler.ToolChangeReq := FALSE;
                ELSIF #fbRecipeHandler.ToolReqNumber = #CurrentTool THEN
                    // Requested tool already in position (e.g. home = slot 1) - skip retract/rotate/extend
                    #fbRecipeHandler.ToolChangeReq := FALSE;
                ELSE
                    #activeToolReq    := #fbRecipeHandler.ToolReqNumber;
                    #bStartSeq        := FALSE;
                    // Release lock before rotating turret: wait T#2S in LOCK_RETRACT_WAIT,
                    // then proceed to STATE_TOOL_CHANGE.
                    #bLockAfterHoming := FALSE;  // LOCK_RETRACT_WAIT exits to STATE_TOOL_CHANGE
                    #State            := STATE_LOCK_RETRACT_WAIT;
                END_IF;
            END_IF;

            // Spindle control from recipe
            IF #fbRecipeHandler.SpindleReqStart THEN
                IF #bSpindleDecelWait THEN
                    // Decel timer still running — capture for deferred apply
                    #bSpindlePendingStart := TRUE;
                    #pendingSpindleSpeed  := #fbRecipeHandler.SpindleReqSpeed;
                ELSE
                    #bSpindleStart := TRUE;
                    "DB_Spindle".Cmd_SetSpeed := #fbRecipeHandler.SpindleReqSpeed;
                END_IF;
            END_IF;
            IF #fbRecipeHandler.SpindleReqStop THEN
                #bSpindleStart       := FALSE;  // Drop RunCmd level
                #bSpindleDecelWait   := TRUE;   // Start decel wait
                #bSpindlePendingStart := FALSE; // Cancel any previous pending start
            END_IF;

            // Complete
            IF #fbRecipeHandler.Done THEN
                #State := 100;  // Go to COMPLETE state, not IDLE
                "DB_HMI".ProgressPercent := 100.0;
                #bSpindleStart := FALSE;  // Drop RunCmd level on completion
                #timerRunning := FALSE; // Stop cycle timer
                #savedLineIndex := -1;  // Clear saved position
                #savedProgram := -1;
                // Arm the end-of-program sanding dwell (2026-08-29). This is the ONLY place
                // it is armed, and State := 100 is assigned nowhere else, so the dwell runs
                // exactly once per completed program -- it cannot re-trigger while the
                // machine sits in COMPLETE. Both config values must be > 0: SandTime_s is
                // the operator's on/off switch, and a SandSpeed of 0 would otherwise be
                // clamped up to MinSpeed and start the spindle at a speed nobody asked for.
                //
                // Tested against the CLAMPED seconds, not the raw config value: a negative
                // SandTime_s typed by mistake must read as "off", and #sandTimeSec has
                // already floored it at 0. Testing the raw value would arm the dwell on a
                // negative number and then run it with PT = T#0S.
                #bSandActive := (#sandTimeSec > 0)
                                AND ("DB_MachineConfig".SandSpeed > 0.0);
            END_IF;

            // Error
            IF #fbRecipeHandler.Error THEN
                #State := STATE_ERROR;
                #newErrorFlag := TRUE;
                #newErrorCode := #fbRecipeHandler.ErrorID;
            END_IF;

        // -----------------------------------------------------------------
        // === STATE_LOCK_EXTEND_WAIT (17) ===
        // -----------------------------------------------------------------
        17: // LOCK_EXTEND_WAIT -- commanding ToolHeadLock to extend; sensor must confirm before RUNNING
            // Cmd_Extend=TRUE is driven outside the CASE (see ToolHeadLock section below).
            // No timer fallback -- lock MUST be confirmed by sensor before machining starts.

 	     #StatusID := 17;
	      IF "DB_HMI".Bypass_ToolHeadLock THEN
	         // Bypass: no sensor wait -- advance immediately (cylinder still commanded to
	         // extend outside the CASE if physically present, but AtSetpoint is not required).
	         #State := STATE_RUNNING;
	      ELSIF "DB_Cylinder_ToolHeadLock".AtSetpoint THEN
 	         #State := STATE_RUNNING;
 	     ELSIF "DB_Cylinder_ToolHeadLock".Error THEN
  	        // Sensor did not confirm within Timeout_Extend (T#3S) — abort
  	        #newErrorFlag := TRUE;
  	        #newErrorCode := 16#0012;
  	        "DB_Diagnostic".Error_Text := 'LockExtendWait: CylFB.Error=TRUE, AtSetpoint=FALSE - check air supply and magnetic sensor';
   	       "DB_HMI".ErrorDetail    := 'Lock sensor (AtSetpoint) not confirmed - check cylinder/sensor';
   	       #State := STATE_ERROR;
   	   END_IF;

        // -----------------------------------------------------------------
        // === STATE_LOCK_RETRACT_WAIT (29) ===
        // -----------------------------------------------------------------
        29: // LOCK_RETRACT_WAIT -- ToolHeadLock releasing (spring return); wait T#2S before proceeding
            // Cmd_Extend=FALSE here (state not RUNNING/PAUSED/LOCK_EXTEND_WAIT); spring retracts.
            // No sensor yet: proceed after timeout regardless.
            // bLockAfterHoming selects exit:
            //   TRUE  = coming from STOPPING → go to STATE_STOPPED (axes already parked at SheetLoadPos)
            //   FALSE = coming from RUNNING (tool change) → go to STATE_TOOL_CHANGE
            #StatusID := 29;
            IF #tonLockWait.Q THEN
                IF #bLockAfterHoming THEN
                    #State := STATE_STOPPED;  // Axes already parked at SheetLoadPos by STOPPING; no homing needed
                ELSE
                    #State := STATE_TOOL_CHANGE;
                END_IF;
            END_IF;

        // -----------------------------------------------------------------
        // === STATE_STOPPING (18) ===
        // -----------------------------------------------------------------
        18: // STOPPING - Stop program without generating an error.
            // Phase 1: recipe executor halts → command spindle stop → start axis park move.
            // Axes move to SheetLoadPos_X/Z (MC_MoveAbsolute, rapid, both simultaneously) in
            // parallel with the spindle decel wait. Target is the sheet-load park, not 0,0:
            // an abort leaves the machine in the same place a normal cycle end does, so the
            // next Start can take the fast path instead of paying for a homing cycle.
            // Phase 2: release MandrelLock once BOTH spindle timer elapsed AND axes done → LOCK_RETRACT_WAIT → STOPPED.
            #StatusID := 18;
            #Running := FALSE;
            #timerRunning := FALSE;
            // Axis return completion check — runs BEFORE the start-trigger so that a stale
            // Done latch from the previous stop cycle (FB_Axis_AbsPos holds Done after Execute
            // drops) cannot immediately cancel bStopMoveX/Z on the same scan they are set.
            // When this check runs first, bStopMoveX/Z are still FALSE on the first scan of
            // STOPPING (no action), and the start-trigger below then sets them correctly.
            //
            // ITEM-56c (2026-08-16): Done and Error used to share one branch, so an axis that
            // FAILED to reach the park cleared its flag exactly as if it had arrived -- no alarm,
            // no ErrorDetail, and the machine reported a clean stop with an axis left wherever the
            // fault dropped it. STATE_STOP_GOTOZERO (21) has always raised 16#0001 / 16#0002 for
            // the identical failure, so the two stop paths disagreed. They now match.
            //
            // Not a safety change: on a variant that HAS a MandrelLock, it is deliberately left
            // EXTENDED on this path. Phase 2 below is the only thing that releases it, and going to
            // STATE_ERROR skips it, so the sheet stays clamped while the spindle coasts down; the
            // operator's Ack then releases it through the ITEM-32 deferred path.
            // On THIS machine there is no MandrelLock cylinder -- the sheet is clamped manually --
            // so that consideration does not apply here either way.
            IF #bStopMoveX THEN
                IF #fbMoveX_Stop.Done THEN
                    #bStopMoveX := FALSE;
                ELSIF #fbMoveX_Stop.Error THEN
                    #bStopMoveX := FALSE;
                    #bStopMoveZ := FALSE;   // drop the sibling Execute too -- STATE_ERROR kills
                                            // drive power anyway, so its move cannot complete
                    #newErrorFlag := TRUE;
                    #newErrorCode := 16#0001;  // X move failed
                    "DB_HMI".ErrorDetail := CONCAT(
                        IN1 := 'X could not reach sheet-load park on stop. TO:',
                        IN2 := "FC_TO_ErrorText"(Code := #fbMoveX_Stop.ErrorID));
                    "DB_Diagnostic".Error_Text :=
                        'STOPPING: X park move failed - axis left short of SheetLoadPos_X';
                    #State := STATE_ERROR;
                END_IF;
            END_IF;
            // Z is checked only while the state is still STOPPING: if X just failed, its report
            // stays on the HMI rather than being overwritten by a second one in the same scan.
            IF #bStopMoveZ AND (#State = STATE_STOPPING) THEN
                IF #fbMoveZ_Stop.Done THEN
                    #bStopMoveZ := FALSE;
                ELSIF #fbMoveZ_Stop.Error THEN
                    #bStopMoveX := FALSE;
                    #bStopMoveZ := FALSE;
                    #newErrorFlag := TRUE;
                    #newErrorCode := 16#0002;  // Z move failed
                    "DB_HMI".ErrorDetail := CONCAT(
                        IN1 := 'Z could not reach sheet-load park on stop. TO:',
                        IN2 := "FC_TO_ErrorText"(Code := #fbMoveZ_Stop.ErrorID));
                    "DB_Diagnostic".Error_Text :=
                        'STOPPING: Z park move failed - axis left short of SheetLoadPos_Z';
                    #State := STATE_ERROR;
                END_IF;
            END_IF;
            // Phase 1: wait for recipe executor to finish, then command spindle stop and
            // begin waiting for the spindle to reach zero speed before releasing MandrelLock.
            // MandrelLock stays extended (sheet clamped) while the spindle decelerates --
            // retracting while spinning could throw the sheet at the operator.
            //
            // The `#State = STATE_STOPPING` term (added with ITEM-56c) is what stops this block
            // from re-arming the park move in the SAME scan that the completion check above sent
            // the machine to STATE_ERROR: that check clears bStopMoveX/Z, which is exactly the
            // condition phase 1 looks for. Same pattern STATE_STOP_GOTOZERO already uses at its
            // own exit test. Do not drop it.
            IF NOT #fbRecipeHandler.Busy AND NOT #bWaitingSpindleStop
               AND (#State = STATE_STOPPING) THEN
                #bSpindleStop             := TRUE;
                #bSheetHolderRetractHold  := TRUE;  // Held: release sheet holder (may be extended if stopped during SHEET_WAIT Ph1/2)
                #bSheetWaitPhase2         := FALSE;
                #bSheetWaitPhase3         := FALSE;
                // ITEM-28: capture commanded speed before issuing stop; compute proportional wait time.
                // Cmd_SetSpeed holds the VFD setpoint from the previous scan (FB_SpindleControl not yet called this scan).
                #capturedSpindleRPM := "DB_Spindle".Cmd_SetSpeed;
                IF "DB_MachineConfig".SpindleMaxRPM > 0.0 THEN
                    #spindleStopPT := DINT_TO_TIME(
                        REAL_TO_DINT(
                            DINT_TO_REAL(TIME_TO_DINT("DB_MachineConfig".SpindleStopSafeTime))
                            * (#capturedSpindleRPM / "DB_MachineConfig".SpindleMaxRPM)
                        )
                    );
                ELSE
                    #spindleStopPT := "DB_MachineConfig".SpindleStopSafeTime;  // safe fallback if MaxRPM not configured
                END_IF;
                #bWaitingSpindleStop := TRUE;   // Enable phase 2 (proportional spindle decel wait)
                // fbMoveX/Z_Stop called at bottom of FB with Execute := bStopMoveX/Z,
                // target parkTargetX/Z (= clamped SheetLoadPos) at RapidVelocity.
                // Both axes start simultaneously.
                #bStopMoveX          := TRUE;   // Start X park move immediately (parallel with spindle decel and Z)
                #bStopMoveZ          := TRUE;   // Start Z park move simultaneously with X
            END_IF;
            // Phase 2: release MandrelLock once proportional spindle decel timer has elapsed AND axes are parked.
            // Bypass_MandrelLock: no cylinder on this variant — skip decel wait, go directly to LOCK_RETRACT_WAIT.
            // No physical encoder -- ActualSpeed is a TO estimate only. tonSpindleStopWait is sole release condition.
            // `#State = STATE_STOPPING` (added with ITEM-56c): without it, a park move that failed
            // above would clear bStopMoveX/Z and this block would then release the MandrelLock and
            // transition to LOCK_RETRACT_WAIT in the same scan -- overwriting the STATE_ERROR that
            // was just set, and unclamping the sheet on a machine with a faulted axis.
            IF #bWaitingSpindleStop AND NOT #bStopMoveX AND NOT #bStopMoveZ
               AND (#State = STATE_STOPPING)
               AND ("DB_MachineConfig".Bypass_MandrelLock OR #tonSpindleStopWait.Q) THEN
                IF NOT "DB_MachineConfig".Bypass_MandrelLock THEN
                    "DB_Cylinder_MandrelLock".Cmd_Extend := FALSE;
                    #bMandrelRetractPulse := TRUE;  // One-shot: release mandrel lock
                END_IF;
                #bWaitingSpindleStop   := FALSE;
                #bLockAfterHoming      := TRUE;  // LOCK_RETRACT_WAIT exits to STATE_STOPPED
                #State                 := STATE_LOCK_RETRACT_WAIT;
            END_IF;

        // -----------------------------------------------------------------
        // === STATE_STOP_GOHOME (19) ===
        // -----------------------------------------------------------------
        19: // STOP_GOHOME - Active homing after stop (X then Z, sequential)
            // BUG FIX: Previous implementation homed X and Z simultaneously.
            // Using the same sequential pattern as STATE_HOMING: X first, then Z.
            #StatusID := 19;
            #Running := FALSE;
            IF #homeSeqState = 1 THEN
                // X homing
                #bHomeXExec := TRUE;
                #bHomeZExec := FALSE;
                IF #fbHomeX.Done THEN
                    #bHomeXExec := FALSE;
                    #homeSeqState := 2;
                    #bHomeZExec := TRUE;
                ELSIF #fbHomeX.Error THEN
                    #bHomeXExec := FALSE;
                    #homeSeqState := 0;
                    #State := STATE_ERROR;
                    #newErrorFlag := TRUE;
                    #newErrorCode := 16#0003;
                    "DB_Diagnostic".HomeX_ErrorID := #fbHomeX.ErrorID;
                    "DB_Diagnostic".TO_ErrorText  := "FC_TO_ErrorText"(Code := #fbHomeX.ErrorID);
                    "DB_HMI".ErrorDetail    := CONCAT(IN1 := 'TO:', IN2 := "DB_Diagnostic".TO_ErrorText);
                END_IF;
            ELSIF #homeSeqState = 2 THEN
                // Z homing
                #bHomeXExec := FALSE;
                #bHomeZExec := TRUE;
                IF #fbHomeZ.Done THEN
                    #bHomeZExec := FALSE;
                    IF NOT "DB_MachineConfig".Bypass_ToolAxis THEN
                        // Proceed to tool axis homing (step 3)
                        #homeSeqState := 3;
                        #bHomeToolExec := TRUE;
                    ELSE
                        // Tool axis bypassed -- homing complete
                        #homeSeqState := 0;
                        #State := STATE_STOPPED;
                    END_IF;
                ELSIF #fbHomeZ.Error THEN
                    #bHomeZExec := FALSE;
                    #homeSeqState := 0;
                    #State := STATE_ERROR;
                    #newErrorFlag := TRUE;
                    #newErrorCode := 16#0004;
                    "DB_Diagnostic".HomeZ_ErrorID := #fbHomeZ.ErrorID;
                    "DB_Diagnostic".TO_ErrorText  := "FC_TO_ErrorText"(Code := #fbHomeZ.ErrorID);
                    "DB_HMI".ErrorDetail    := CONCAT(IN1 := 'TO:', IN2 := "DB_Diagnostic".TO_ErrorText);
                END_IF;
            ELSIF #homeSeqState = 3 THEN
                // Homing Tool axis
                #bHomeToolExec := TRUE;
                IF #fbHomeTool.Done THEN
                    #bHomeToolExec := FALSE;
                    #homeSeqState := 0;
                    #State := STATE_STOPPED;
                ELSIF #fbHomeTool.Error THEN
                    #bHomeToolExec := FALSE;
                    #homeSeqState := 0;
                    #State := STATE_ERROR;
                    #newErrorFlag := TRUE;
                    #newErrorCode := 16#0007;
                    "DB_Diagnostic".HomeTool_ErrorID := #fbHomeTool.ErrorID;
                    "DB_Diagnostic".TO_ErrorText     := "FC_TO_ErrorText"(Code := #fbHomeTool.ErrorID);
                    "DB_HMI".ErrorDetail    := CONCAT(IN1 := 'TO:', IN2 := "DB_Diagnostic".TO_ErrorText);
                END_IF;
            ELSE
                // homeSeqState invalid -- safe fallback
                #homeSeqState := 0;
                #bHomeXExec := FALSE;
                #bHomeZExec := FALSE;
                #bHomeToolExec := FALSE;
                #State := STATE_STOPPED;
            END_IF;
            // ITEM-30: independent 120s timeout for STATE_STOP_GOHOME (tonStopHomeTimeout)
            // Previously used tonHomingTimeout which could be nearly exhausted by a preceding STATE_HOMING run.
            IF #tonStopHomeTimeout.Q THEN
                #bHomeXExec := FALSE;
                #bHomeZExec := FALSE;
                #bHomeToolExec := FALSE;
                #homeSeqState := 0;
                #State := STATE_ERROR;
                #newErrorFlag := TRUE;
                #newErrorCode := 16#000B;
                "DB_HMI".ErrorDetail    := 'Post-stop homing did not complete - check reference switch/drive';
            END_IF;

        // -----------------------------------------------------------------
        // === STATE_STOP_GOTOZERO (21) ===
        // -----------------------------------------------------------------
        21: // STOP_GOTOZERO - Go to position 0 after stop
            #StatusID := 21;
            #Running := FALSE;
            // Has X axis motion completed?
            IF #bStopMoveX AND #fbMoveX_Stop.Done THEN
                #bStopMoveX := FALSE;
            ELSIF #bStopMoveX AND #fbMoveX_Stop.Error THEN
                #bStopMoveX := FALSE;
                #State := STATE_ERROR;
                #newErrorFlag := TRUE;
                #newErrorCode := 16#0001; // X move failed
                "DB_HMI".ErrorDetail    := 'X axis could not return to zero after stop';
            END_IF;
            // Has Z axis motion completed?
            IF #bStopMoveZ AND #fbMoveZ_Stop.Done THEN
                #bStopMoveZ := FALSE;
            ELSIF #bStopMoveZ AND #fbMoveZ_Stop.Error THEN
                #bStopMoveZ := FALSE;
                #State := STATE_ERROR;
                #newErrorFlag := TRUE;
                #newErrorCode := 16#0002; // Z move failed
                "DB_HMI".ErrorDetail    := 'Z axis could not return to zero after stop';
            END_IF;
            // When both axes are done, return to STOPPED
            IF NOT #bStopMoveX AND NOT #bStopMoveZ AND (#State = STATE_STOP_GOTOZERO) THEN
                #State := STATE_STOPPED;
            END_IF;

        // -----------------------------------------------------------------
        // === STATE_PNP_HALT (22) ===
        // -----------------------------------------------------------------
        22: // PNP_HALT -- axis halted at proximity zone; drives ON, reverse jog allowed to escape
            #StatusID := 22;
            #Running := FALSE;
            // Auto-exit: PNP zone cleared (axis has moved away) -- return to STOPPED
            IF NOT #HW_PNP_X_Min AND NOT #HW_PNP_X_Max THEN #bHaltX_PNP := FALSE; END_IF;
            IF NOT #HW_PNP_Z_Min AND NOT #HW_PNP_Z_Max THEN #bHaltZ_PNP := FALSE; END_IF;
            IF NOT #bHaltX_PNP AND NOT #bHaltZ_PNP THEN
                // ITEM-56h (2026-08-16): acknowledge the alarm here too. The machine state and the
                // alarm are separate -- clearing one does not clear the other. This exit set
                // State := STOPPED but told FB_AlarmManager nothing, so 16#0121..0124 stayed ACTIVE
                // in DB_Error and the HMI showed a live red alarm on a machine reading "Stopped".
                // The operator then had to press Reset purely to clear the red, on a machine that
                // had already recovered by itself -- which is how operators learn to distrust
                // alarms. The manual exit below has always done this; the two now match.
                //
                // Reachable in practice: MC_Halt decelerates, so the axis can come to rest right at
                // the EDGE of the detection zone and vibration flickers the sensor FALSE.
                #Error := FALSE;
                #fbAlarmManager(NewError := FALSE, NewErrorCode := 0, AcknowledgeError := TRUE);
                #State := STATE_STOPPED;
            END_IF;
            // Manual exit: operator presses AckError or Reset
            IF (#ackEdge OR #fbInputs.Cmd_Reset) AND (#EStop_OK OR "DB_HMI".Bypass_EStop) THEN
                #bHaltX_PNP := FALSE;
                #bHaltZ_PNP := FALSE;
                #Error := FALSE;
                #prevSafetyError := FALSE;
                #fbAlarmManager(NewError := FALSE, NewErrorCode := 0, AcknowledgeError := TRUE);
                #State := STATE_STOPPED;
            END_IF;
            // Forward spindle commands from recipe handler.
            // When PNP fires during STATE_RUNNING, the RUNNING(20) case is skipped, so
            // bSpindleStart is never updated from fbRecipeHandler signals. Mirror them here.
            // Note: fbRecipeHandler runs AFTER this CASE, so values here are from previous scan.
            IF #fbRecipeHandler.SpindleReqStop THEN
                #bSpindleStart := FALSE;  // Drop RunCmd level
            END_IF;
            IF #fbRecipeHandler.SpindleReqStart THEN
                #bSpindleStart := TRUE;
                "DB_Spindle".Cmd_SetSpeed := #fbRecipeHandler.SpindleReqSpeed;
            END_IF;

        // -----------------------------------------------------------------
        // === STATE_PAUSED (25) ===
        // -----------------------------------------------------------------
        25: // PAUSED
            #StatusID := 88;
            // Stop elapsed time counting while paused
            #timerRunning := FALSE;
            // Spindle is stopped while paused (RunCmd gated off below on State=PAUSED
            // when NOT bResumeSpeedup). On Continue the resume runs in TWO phases:
            //   Phase 1 (bResumeLockChk) → confirm the ToolHeadLock is actually engaged
            //   Phase 2 (bResumeSpeedup) → restart the spindle and wait
            //                              SpindleResumeSpeedupTime for it to reach speed
            //                              BEFORE releasing the axes
            // bPauseActive stays TRUE across BOTH phases → FB_RecipeHandler holds at the
            // retract point (802). When the spin-up timer elapses, drop bPauseActive →
            // FB_RecipeHandler returns to the interruption point (803) and machining resumes.
            // Only Btn_Continue resumes (Pause button does NOT toggle).
            IF #continueEdge THEN
                #bResumeLockChk := TRUE;
            END_IF;

